TYPE FaultHandling :
STRUCT
    FaultID : int;
END_STRUCT
END_TYPE

(* stored: Version 1.1.0.1, ProductVersion 3.1.4024.12
   DUT FaultHandling: Id {27f899fe-1bd5-0745-1765-7b65e27419c1} *)
